// TIA Portal V17 export
// export: Created 2025-06-26T07:49:38.9471019Z, ExportSetting WithDefaults, DisplayName Totally Integrated Automation Portal, DisplayVersion V17 Update 8, DisplayName TIA Portal Openness, DisplayVersion V17 Update 8, DisplayName TIA Portal Version Control Interface, DisplayVersion V17, DisplayName STEP 7 Professional, DisplayVersion V17 Update 8, DisplayName STEP 7 Safety, DisplayVersion V17 Update 6, DisplayName WinCC Advanced, DisplayVersion V17 Update 8
FUNCTION_BLOCK "ControlAlarmHandling"   // FB19, FBD
{ S7_Optimized_Access := 'TRUE' }
VERSION : 0.1
// stored: AutoNumber true, IsIECCheckEnabled false, IsRetainMemResEnabled false, MemoryReserve 0, SetENOAutomatically false, UDAEnableTagReadback false
   VAR
      A1004 { ExternalAccessible := 'False'; ExternalVisible := 'False'; ExternalWritable := 'False'; S7_SetPoint := 'True'} : "fbHMIEvent";
      A2018 { ExternalAccessible := 'False'; ExternalVisible := 'False'; ExternalWritable := 'False'; S7_SetPoint := 'True'} : "fbHighAlarm";
      A2028 { ExternalAccessible := 'False'; ExternalVisible := 'False'; ExternalWritable := 'False'; S7_SetPoint := 'True'} : "fbLowAlarm";
      A2058 { ExternalAccessible := 'False'; ExternalVisible := 'False'; ExternalWritable := 'False'; S7_SetPoint := 'True'} : "fbLowAlarm";
      A2100 { ExternalAccessible := 'False'; ExternalVisible := 'False'; ExternalWritable := 'False'; S7_SetPoint := 'True'} : "fbHighAlarm";
      A2101 { ExternalAccessible := 'False'; ExternalVisible := 'False'; ExternalWritable := 'False'; S7_SetPoint := 'True'} : "fbHighAlarm";
      A2102 { ExternalAccessible := 'False'; ExternalVisible := 'False'; ExternalWritable := 'False'; S7_SetPoint := 'True'} : "fbHighAlarm";
      A2103 { ExternalAccessible := 'False'; ExternalVisible := 'False'; ExternalWritable := 'False'; S7_SetPoint := 'True'} : "fbHighAlarm";
      A2105 { ExternalAccessible := 'False'; ExternalVisible := 'False'; ExternalWritable := 'False'; S7_SetPoint := 'True'} : "fbHighAlarm";
      A2106 { ExternalAccessible := 'False'; ExternalVisible := 'False'; ExternalWritable := 'False'; S7_SetPoint := 'True'} : "fbHighAlarm";
      A2107 { ExternalAccessible := 'False'; ExternalVisible := 'False'; ExternalWritable := 'False'; S7_SetPoint := 'True'} : "fbHighAlarm";
      A2109 { ExternalAccessible := 'False'; ExternalVisible := 'False'; ExternalWritable := 'False'; S7_SetPoint := 'True'} : "fbHighAlarm";
      A2108 { ExternalAccessible := 'False'; ExternalVisible := 'False'; ExternalWritable := 'False'; S7_SetPoint := 'True'} : "fbHighAlarm";
      A2110 { ExternalAccessible := 'False'; ExternalVisible := 'False'; ExternalWritable := 'False'; S7_SetPoint := 'True'} : "fbHighAlarm";
      A2111 { ExternalAccessible := 'False'; ExternalVisible := 'False'; ExternalWritable := 'False'; S7_SetPoint := 'True'} : "fbHighAlarm";
      A2112 { ExternalAccessible := 'False'; ExternalVisible := 'False'; ExternalWritable := 'False'; S7_SetPoint := 'True'} : "fbHighAlarm";
      A2113 { ExternalAccessible := 'False'; ExternalVisible := 'False'; ExternalWritable := 'False'; S7_SetPoint := 'True'} : "fbHighAlarm";
      A2114 { ExternalAccessible := 'False'; ExternalVisible := 'False'; ExternalWritable := 'False'; S7_SetPoint := 'True'} : "fbHighAlarm";
      A2115 { ExternalAccessible := 'False'; ExternalVisible := 'False'; ExternalWritable := 'False'; S7_SetPoint := 'True'} : "fbLowAlarm";
      A2116 { ExternalAccessible := 'False'; ExternalVisible := 'False'; ExternalWritable := 'False'; S7_SetPoint := 'True'} : "fbHighAlarm";
      A2117 { ExternalAccessible := 'False'; ExternalVisible := 'False'; ExternalWritable := 'False'; S7_SetPoint := 'True'} : "fbLowAlarm";
      A2301 { ExternalAccessible := 'False'; ExternalVisible := 'False'; ExternalWritable := 'False'; S7_SetPoint := 'True'} : "fbLowAlarm";
      A2302 { ExternalAccessible := 'False'; ExternalVisible := 'False'; ExternalWritable := 'False'; S7_SetPoint := 'True'} : "fbHighAlarm";
      A2303 { ExternalAccessible := 'False'; ExternalVisible := 'False'; ExternalWritable := 'False'; S7_SetPoint := 'True'} : "fbHighAlarm";
      A2304 { ExternalAccessible := 'False'; ExternalVisible := 'False'; ExternalWritable := 'False'; S7_SetPoint := 'True'} : "fbLowAlarm";
      A2305 { ExternalAccessible := 'False'; ExternalVisible := 'False'; ExternalWritable := 'False'; S7_SetPoint := 'True'} : "fbHighAlarm";
      A2306 { ExternalAccessible := 'False'; ExternalVisible := 'False'; ExternalWritable := 'False'; S7_SetPoint := 'True'} : "fbHighAlarm";
      A2307 { ExternalAccessible := 'False'; ExternalVisible := 'False'; ExternalWritable := 'False'; S7_SetPoint := 'True'} : "fbHMIEvent";
      A2308 { ExternalAccessible := 'False'; ExternalVisible := 'False'; ExternalWritable := 'False'; S7_SetPoint := 'True'} : "fbHighAlarm";
      A3400 { ExternalAccessible := 'False'; ExternalVisible := 'False'; ExternalWritable := 'False'; S7_SetPoint := 'True'} : "fbHMIEvent";
      A9023 { ExternalAccessible := 'False'; ExternalVisible := 'False'; ExternalWritable := 'False'; S7_SetPoint := 'True'} : "fbDeviationAlarm";
      A9024 { S7_SetPoint := 'True'} : "fbDeviationAlarm";
      A9025 { S7_SetPoint := 'True'} : "fbDeviationAlarm";
      A9026 { S7_SetPoint := 'True'} : "fbDeviationAlarm";
      A9027 { S7_SetPoint := 'True'} : "fbDeviationAlarm";
      A9028 { S7_SetPoint := 'True'} : "fbDeviationAlarm";
      A9029 { S7_SetPoint := 'True'} : "fbDeviationAlarm";
      A9030 { S7_SetPoint := 'True'} : "fbDeviationAlarm";
      A9031 { S7_SetPoint := 'True'} : "fbDeviationAlarm";
   END_VAR
   VAR_TEMP   // added for the SCL form of the ladder/FBD networks
      _w1 : Bool;
   END_VAR
BEGIN

REGION Network 1: 1004
   // DISABLED when no connection
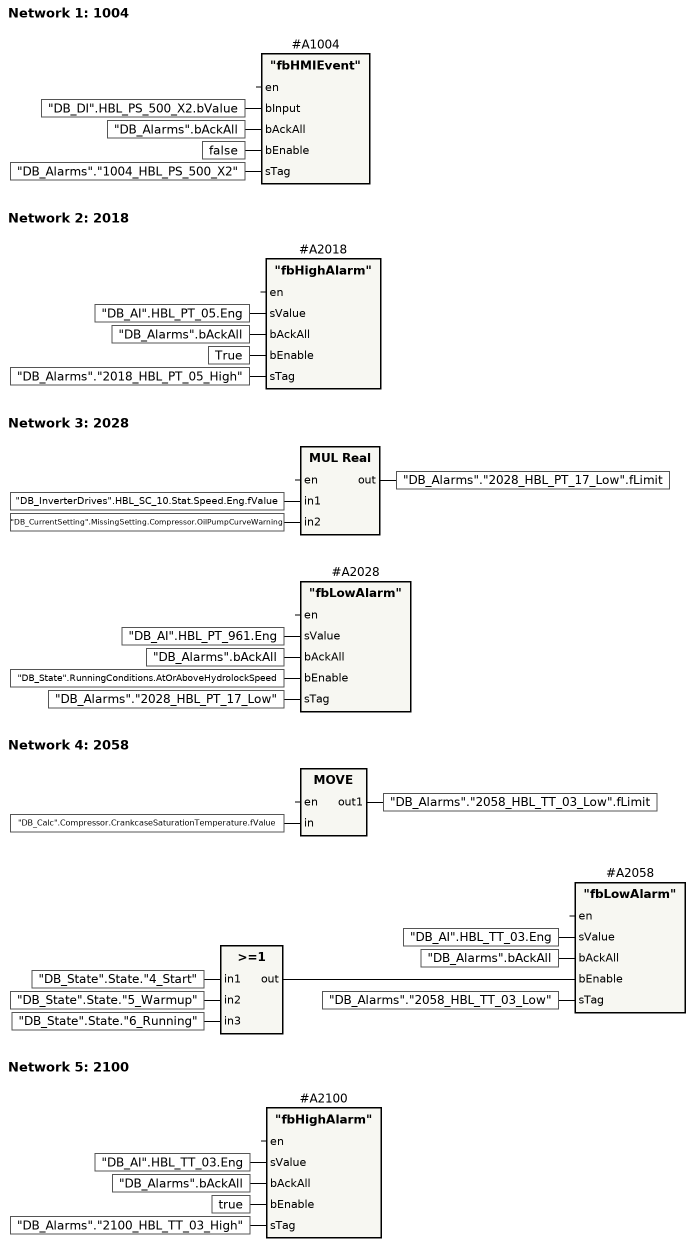
   #A1004(bInput := "DB_DI".HBL_PS_500_X2.bValue,   // "fbHMIEvent"
          bAckAll := "DB_Alarms".bAckAll,
          bEnable := false,
          sTag := "DB_Alarms"."1004_HBL_PS_500_X2");
END_REGION

REGION Network 2: 2018
   #A2018(sValue := "DB_AI".HBL_PT_05.Eng,   // "fbHighAlarm"
          bAckAll := "DB_Alarms".bAckAll,
          bEnable := True,
          sTag := "DB_Alarms"."2018_HBL_PT_05_High");
END_REGION

REGION Network 3: 2028
   // NOTE: alarm limit is dynamic, so don't move it to InitCurrentSettings
   "DB_Alarms"."2028_HBL_PT_17_Low".fLimit := "DB_InverterDrives".HBL_SC_10.Stat.Speed.Eng.fValue * "DB_CurrentSetting".MissingSetting.Compressor.OilPumpCurveWarning;
   #A2028(sValue := "DB_AI".HBL_PT_961.Eng,   // "fbLowAlarm"
          bAckAll := "DB_Alarms".bAckAll,
          bEnable := "DB_State".RunningConditions.AtOrAboveHydrolockSpeed,
          sTag := "DB_Alarms"."2028_HBL_PT_17_Low");
END_REGION

REGION Network 4: 2058
   // NOTE: alarm Low limit is dynamic, so don't move it to InitCurrentSettings
   "DB_Alarms"."2058_HBL_TT_03_Low".fLimit := "DB_Calc".Compressor.CrankcaseSaturationTemperature.fValue;
   #A2058(sValue := "DB_AI".HBL_TT_03.Eng,   // "fbLowAlarm"
          bAckAll := "DB_Alarms".bAckAll,
          bEnable := "DB_State".State."4_Start" OR "DB_State".State."5_Warmup" OR "DB_State".State."6_Running",
          sTag := "DB_Alarms"."2058_HBL_TT_03_Low");
END_REGION

REGION Network 5: 2100
   #A2100(sValue := "DB_AI".HBL_TT_03.Eng,   // "fbHighAlarm"
          bAckAll := "DB_Alarms".bAckAll,
          bEnable := true,
          sTag := "DB_Alarms"."2100_HBL_TT_03_High");
END_REGION

REGION Network 6: 2101
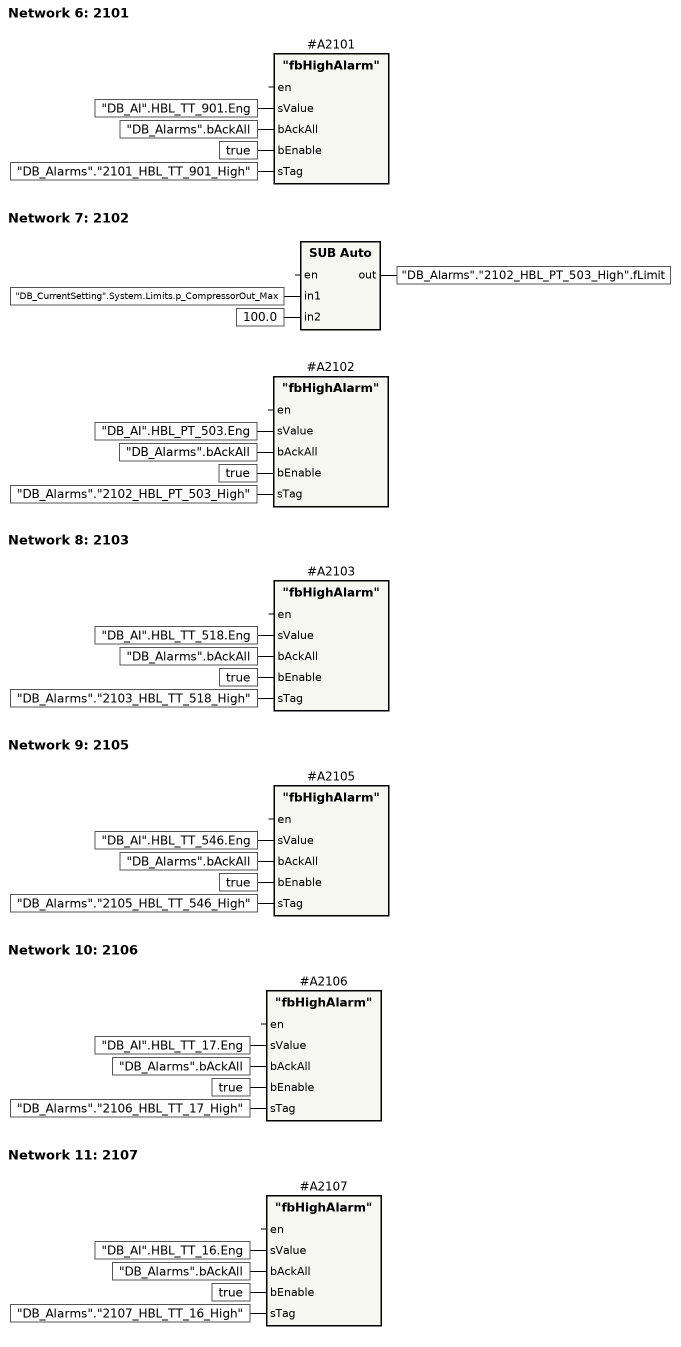
   #A2101(sValue := "DB_AI".HBL_TT_901.Eng,   // "fbHighAlarm"
          bAckAll := "DB_Alarms".bAckAll,
          bEnable := true,
          sTag := "DB_Alarms"."2101_HBL_TT_901_High");
END_REGION

REGION Network 7: 2102
   // Update the alarm limit ALL THE TIME, not just at PLC startup. If the p_CompressorOut_Max value is changed, then this alarms should ALWAYS follow
   "DB_Alarms"."2102_HBL_PT_503_High".fLimit := "DB_CurrentSetting".System.Limits.p_CompressorOut_Max - 100.0;
   #A2102(sValue := "DB_AI".HBL_PT_503.Eng,   // "fbHighAlarm"
          bAckAll := "DB_Alarms".bAckAll,
          bEnable := true,
          sTag := "DB_Alarms"."2102_HBL_PT_503_High");
END_REGION

REGION Network 8: 2103
   #A2103(sValue := "DB_AI".HBL_TT_518.Eng,   // "fbHighAlarm"
          bAckAll := "DB_Alarms".bAckAll,
          bEnable := true,
          sTag := "DB_Alarms"."2103_HBL_TT_518_High");
END_REGION

REGION Network 9: 2105
   #A2105(sValue := "DB_AI".HBL_TT_546.Eng,   // "fbHighAlarm"
          bAckAll := "DB_Alarms".bAckAll,
          bEnable := true,
          sTag := "DB_Alarms"."2105_HBL_TT_546_High");
END_REGION

REGION Network 10: 2106
   #A2106(sValue := "DB_AI".HBL_TT_17.Eng,   // "fbHighAlarm"
          bAckAll := "DB_Alarms".bAckAll,
          bEnable := true,
          sTag := "DB_Alarms"."2106_HBL_TT_17_High");
END_REGION

REGION Network 11: 2107
   #A2107(sValue := "DB_AI".HBL_TT_16.Eng,   // "fbHighAlarm"
          bAckAll := "DB_Alarms".bAckAll,
          bEnable := true,
          sTag := "DB_Alarms"."2107_HBL_TT_16_High");
END_REGION

REGION Network 12: 2108
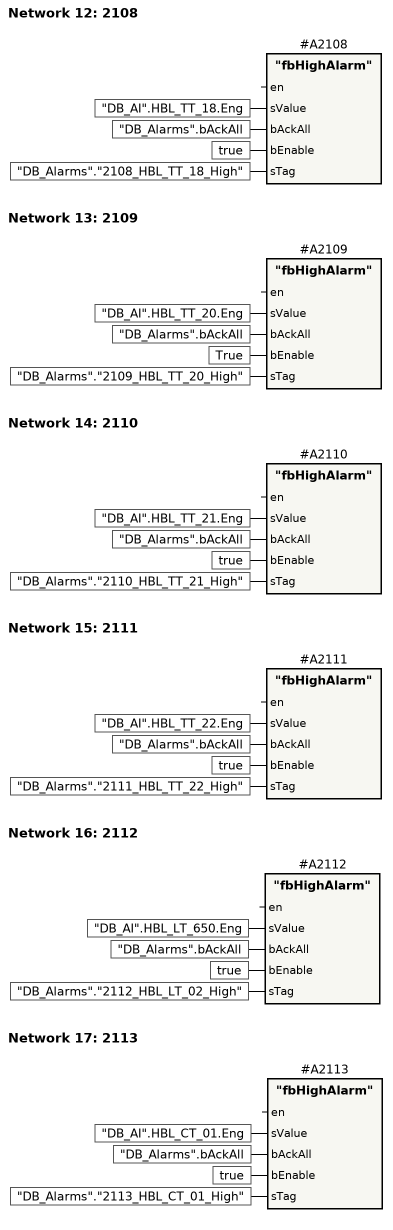
   #A2108(sValue := "DB_AI".HBL_TT_18.Eng,   // "fbHighAlarm"
          bAckAll := "DB_Alarms".bAckAll,
          bEnable := true,
          sTag := "DB_Alarms"."2108_HBL_TT_18_High");
END_REGION

REGION Network 13: 2109
   #A2109(sValue := "DB_AI".HBL_TT_20.Eng,   // "fbHighAlarm"
          bAckAll := "DB_Alarms".bAckAll,
          bEnable := True,
          sTag := "DB_Alarms"."2109_HBL_TT_20_High");
END_REGION

REGION Network 14: 2110
   #A2110(sValue := "DB_AI".HBL_TT_21.Eng,   // "fbHighAlarm"
          bAckAll := "DB_Alarms".bAckAll,
          bEnable := true,
          sTag := "DB_Alarms"."2110_HBL_TT_21_High");
END_REGION

REGION Network 15: 2111
   #A2111(sValue := "DB_AI".HBL_TT_22.Eng,   // "fbHighAlarm"
          bAckAll := "DB_Alarms".bAckAll,
          bEnable := true,
          sTag := "DB_Alarms"."2111_HBL_TT_22_High");
END_REGION

REGION Network 16: 2112
   #A2112(sValue := "DB_AI".HBL_LT_650.Eng,   // "fbHighAlarm"
          bAckAll := "DB_Alarms".bAckAll,
          bEnable := true,
          sTag := "DB_Alarms"."2112_HBL_LT_02_High");
END_REGION

REGION Network 17: 2113
   #A2113(sValue := "DB_AI".HBL_CT_01.Eng,   // "fbHighAlarm"
          bAckAll := "DB_Alarms".bAckAll,
          bEnable := true,
          sTag := "DB_Alarms"."2113_HBL_CT_01_High");
END_REGION

REGION Network 18: 2114
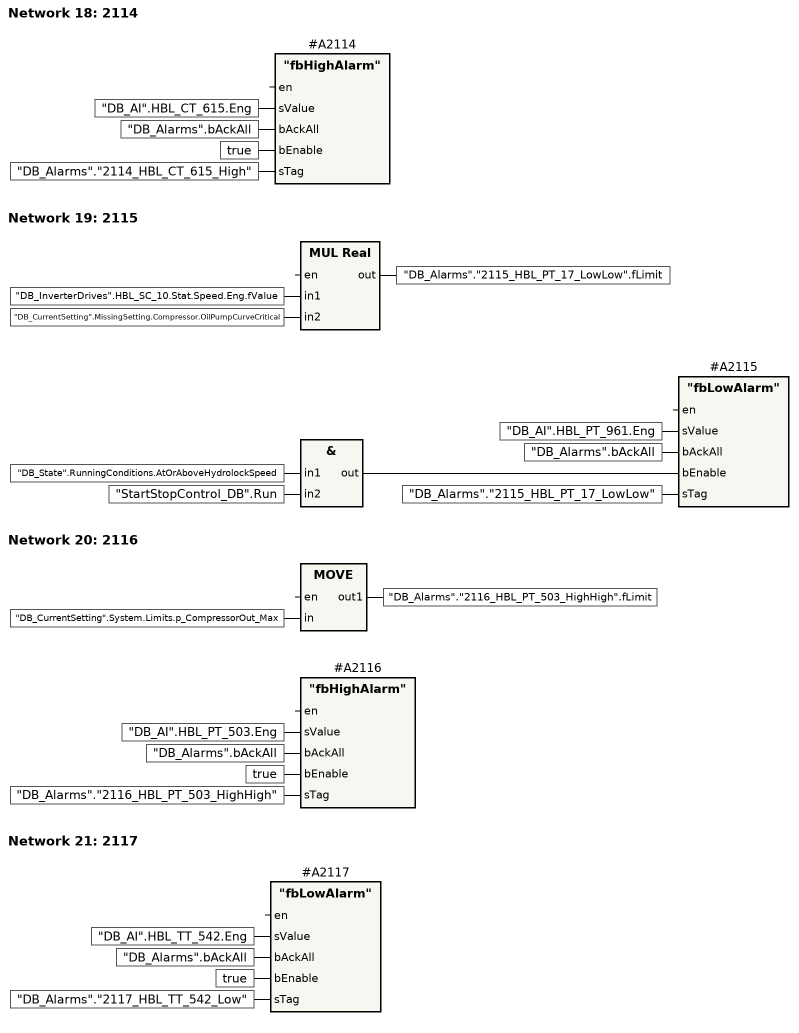
   #A2114(sValue := "DB_AI".HBL_CT_615.Eng,   // "fbHighAlarm"
          bAckAll := "DB_Alarms".bAckAll,
          bEnable := true,
          sTag := "DB_Alarms"."2114_HBL_CT_615_High");
END_REGION

REGION Network 19: 2115
   // NOTE: alarm limit is dynamic, so don't move it to InitCurrentSettings
   "DB_Alarms"."2115_HBL_PT_17_LowLow".fLimit := "DB_InverterDrives".HBL_SC_10.Stat.Speed.Eng.fValue * "DB_CurrentSetting".MissingSetting.Compressor.OilPumpCurveCritical;
   #A2115(sValue := "DB_AI".HBL_PT_961.Eng,   // "fbLowAlarm"
          bAckAll := "DB_Alarms".bAckAll,
          bEnable := "DB_State".RunningConditions.AtOrAboveHydrolockSpeed AND "StartStopControl_DB".Run,
          sTag := "DB_Alarms"."2115_HBL_PT_17_LowLow");
END_REGION

REGION Network 20: 2116
   // Update the alarm limit ALL THE TIME, not just at PLC startup. If the p_CompressorOut_Max value is changed, then this alarms should ALWAYS follow
   "DB_Alarms"."2116_HBL_PT_503_HighHigh".fLimit := "DB_CurrentSetting".System.Limits.p_CompressorOut_Max;
   #A2116(sValue := "DB_AI".HBL_PT_503.Eng,   // "fbHighAlarm"
          bAckAll := "DB_Alarms".bAckAll,
          bEnable := true,
          sTag := "DB_Alarms"."2116_HBL_PT_503_HighHigh");
END_REGION

REGION Network 21: 2117
   #A2117(sValue := "DB_AI".HBL_TT_542.Eng,   // "fbLowAlarm"
          bAckAll := "DB_Alarms".bAckAll,
          bEnable := true,
          sTag := "DB_Alarms"."2117_HBL_TT_542_Low");
END_REGION

REGION Network 22: 2301 & 2302
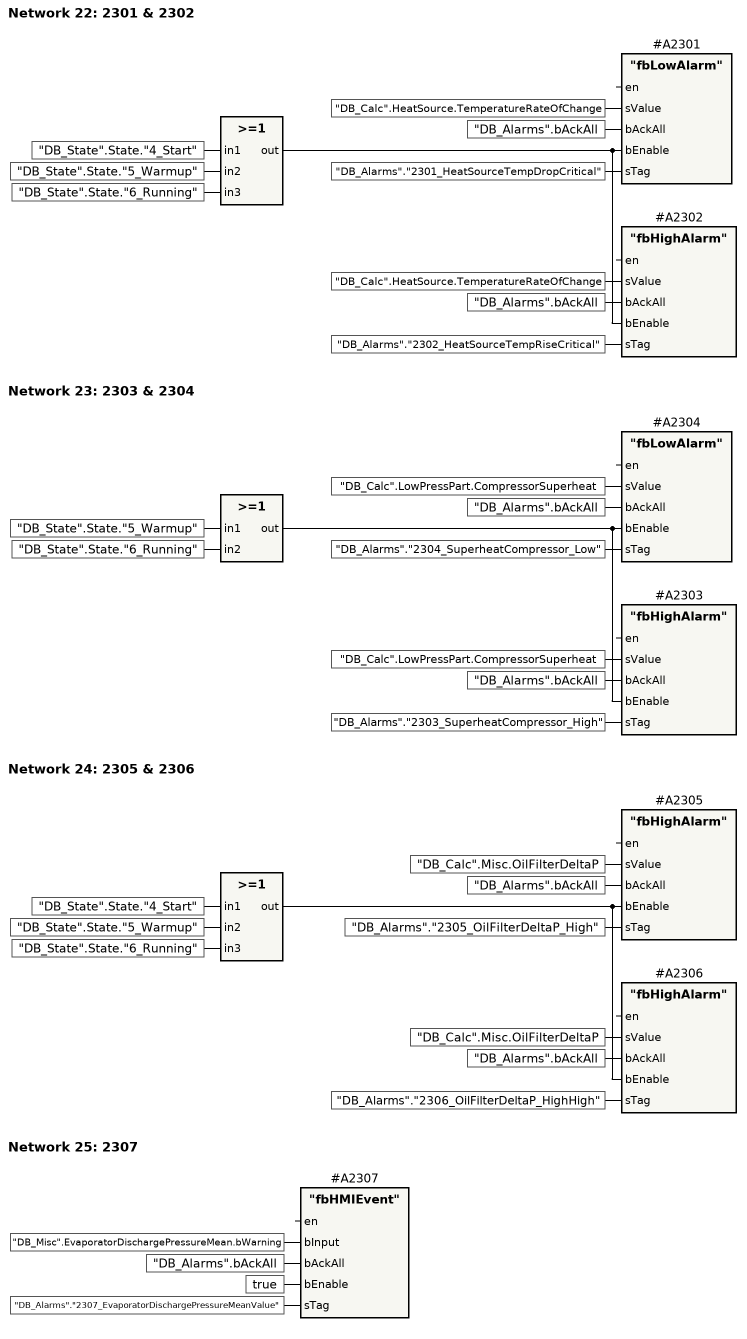
   #_w1 := "DB_State".State."4_Start" OR "DB_State".State."5_Warmup" OR "DB_State".State."6_Running";
   #A2301(sValue := "DB_Calc".HeatSource.TemperatureRateOfChange,   // "fbLowAlarm"
          bAckAll := "DB_Alarms".bAckAll,
          bEnable := #_w1,
          sTag := "DB_Alarms"."2301_HeatSourceTempDropCritical");
   #A2302(sValue := "DB_Calc".HeatSource.TemperatureRateOfChange,   // "fbHighAlarm"
          bAckAll := "DB_Alarms".bAckAll,
          bEnable := #_w1,
          sTag := "DB_Alarms"."2302_HeatSourceTempRiseCritical");
END_REGION

REGION Network 23: 2303 & 2304
   #_w1 := "DB_State".State."5_Warmup" OR "DB_State".State."6_Running";
   #A2304(sValue := "DB_Calc".LowPressPart.CompressorSuperheat,   // "fbLowAlarm"
          bAckAll := "DB_Alarms".bAckAll,
          bEnable := #_w1,
          sTag := "DB_Alarms"."2304_SuperheatCompressor_Low");
   #A2303(sValue := "DB_Calc".LowPressPart.CompressorSuperheat,   // "fbHighAlarm"
          bAckAll := "DB_Alarms".bAckAll,
          bEnable := #_w1,
          sTag := "DB_Alarms"."2303_SuperheatCompressor_High");
END_REGION

REGION Network 24: 2305 & 2306
   #_w1 := "DB_State".State."4_Start" OR "DB_State".State."5_Warmup" OR "DB_State".State."6_Running";
   #A2305(sValue := "DB_Calc".Misc.OilFilterDeltaP,   // "fbHighAlarm"
          bAckAll := "DB_Alarms".bAckAll,
          bEnable := #_w1,
          sTag := "DB_Alarms"."2305_OilFilterDeltaP_High");
   #A2306(sValue := "DB_Calc".Misc.OilFilterDeltaP,   // "fbHighAlarm"
          bAckAll := "DB_Alarms".bAckAll,
          bEnable := #_w1,
          sTag := "DB_Alarms"."2306_OilFilterDeltaP_HighHigh");
END_REGION

REGION Network 25: 2307
   #A2307(bInput := "DB_Misc".EvaporatorDischargePressureMean.bWarning,   // "fbHMIEvent"
          bAckAll := "DB_Alarms".bAckAll,
          bEnable := true,
          sTag := "DB_Alarms"."2307_EvaporatorDischargePressureMeanValue");
END_REGION

REGION Network 26: 2308
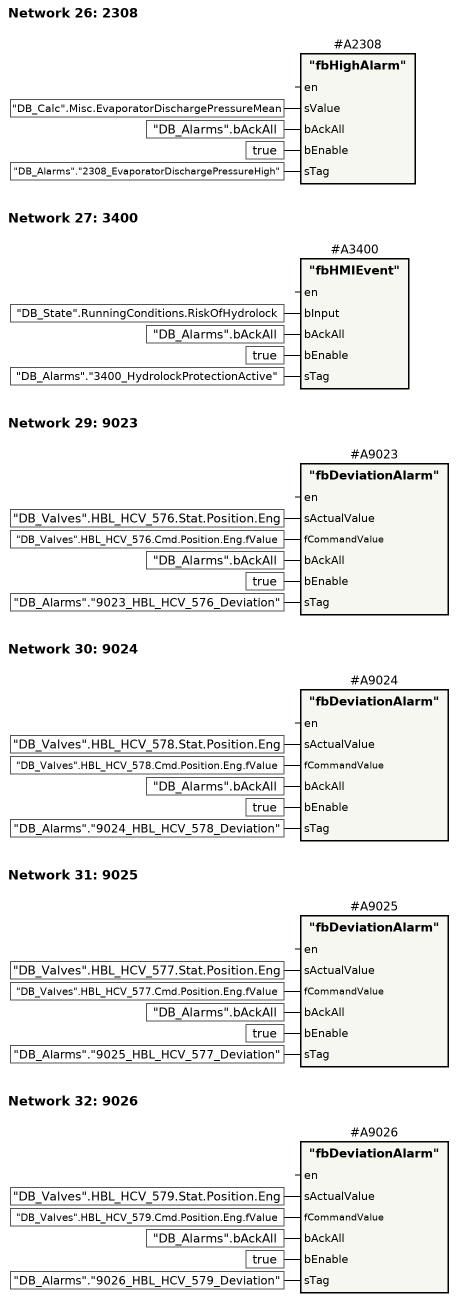
   #A2308(sValue := "DB_Calc".Misc.EvaporatorDischargePressureMean,   // "fbHighAlarm"
          bAckAll := "DB_Alarms".bAckAll,
          bEnable := true,
          sTag := "DB_Alarms"."2308_EvaporatorDischargePressureHigh");
END_REGION

REGION Network 27: 3400
   #A3400(bInput := "DB_State".RunningConditions.RiskOfHydrolock,   // "fbHMIEvent"
          bAckAll := "DB_Alarms".bAckAll,
          bEnable := true,
          sTag := "DB_Alarms"."3400_HydrolockProtectionActive");
END_REGION

REGION Network 28 (SCL): 9023 old
   // This is a deviation alarm, for which a dedicated type does not exist. So we make one here for now with hardocded limits.
   (*
   #A9023(bAckAll := "DB_Alarms".bAckAll, 
           bInput := (ABS(IN := "DB_Valves".HBL_HCV_576.Stat.Position.Eng.fValue -"DB_Valves".HBL_HCV_576.Cmd.Position.Eng.fValue) > 4) OR 
                     ("DB_Valves".HBL_HCV_576.Cmd.Position.Eng.fValue <= 0 AND "DB_Valves".HBL_HCV_576.Stat.Position.Eng.fValue <2),
           sTag := "DB_Alarms"."9023_ExpansionValveDeviation");

   *)
END_REGION

REGION Network 29: 9023
   #A9023(sActualValue := "DB_Valves".HBL_HCV_576.Stat.Position.Eng,   // "fbDeviationAlarm"
          fCommandValue := "DB_Valves".HBL_HCV_576.Cmd.Position.Eng.fValue,
          bAckAll := "DB_Alarms".bAckAll,
          bEnable := true,
          sTag := "DB_Alarms"."9023_HBL_HCV_576_Deviation");
END_REGION

REGION Network 30: 9024
   #A9024(sActualValue := "DB_Valves".HBL_HCV_578.Stat.Position.Eng,   // "fbDeviationAlarm"
          fCommandValue := "DB_Valves".HBL_HCV_578.Cmd.Position.Eng.fValue,
          bAckAll := "DB_Alarms".bAckAll,
          bEnable := true,
          sTag := "DB_Alarms"."9024_HBL_HCV_578_Deviation");
END_REGION

REGION Network 31: 9025
   #A9025(sActualValue := "DB_Valves".HBL_HCV_577.Stat.Position.Eng,   // "fbDeviationAlarm"
          fCommandValue := "DB_Valves".HBL_HCV_577.Cmd.Position.Eng.fValue,
          bAckAll := "DB_Alarms".bAckAll,
          bEnable := true,
          sTag := "DB_Alarms"."9025_HBL_HCV_577_Deviation");
END_REGION

REGION Network 32: 9026
   #A9026(sActualValue := "DB_Valves".HBL_HCV_579.Stat.Position.Eng,   // "fbDeviationAlarm"
          fCommandValue := "DB_Valves".HBL_HCV_579.Cmd.Position.Eng.fValue,
          bAckAll := "DB_Alarms".bAckAll,
          bEnable := true,
          sTag := "DB_Alarms"."9026_HBL_HCV_579_Deviation");
END_REGION

REGION Network 33: 9027
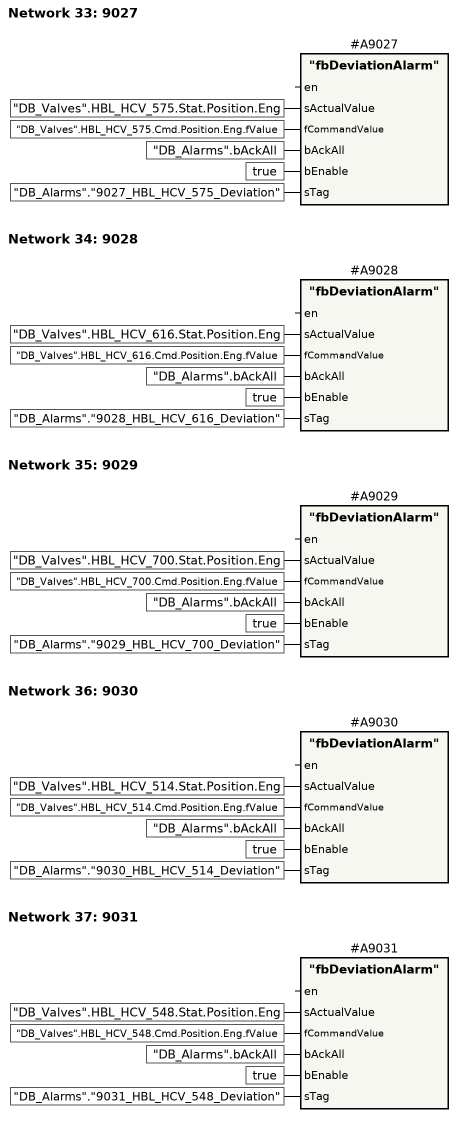
   #A9027(sActualValue := "DB_Valves".HBL_HCV_575.Stat.Position.Eng,   // "fbDeviationAlarm"
          fCommandValue := "DB_Valves".HBL_HCV_575.Cmd.Position.Eng.fValue,
          bAckAll := "DB_Alarms".bAckAll,
          bEnable := true,
          sTag := "DB_Alarms"."9027_HBL_HCV_575_Deviation");
END_REGION

REGION Network 34: 9028
   #A9028(sActualValue := "DB_Valves".HBL_HCV_616.Stat.Position.Eng,   // "fbDeviationAlarm"
          fCommandValue := "DB_Valves".HBL_HCV_616.Cmd.Position.Eng.fValue,
          bAckAll := "DB_Alarms".bAckAll,
          bEnable := true,
          sTag := "DB_Alarms"."9028_HBL_HCV_616_Deviation");
END_REGION

REGION Network 35: 9029
   #A9029(sActualValue := "DB_Valves".HBL_HCV_700.Stat.Position.Eng,   // "fbDeviationAlarm"
          fCommandValue := "DB_Valves".HBL_HCV_700.Cmd.Position.Eng.fValue,
          bAckAll := "DB_Alarms".bAckAll,
          bEnable := true,
          sTag := "DB_Alarms"."9029_HBL_HCV_700_Deviation");
END_REGION

REGION Network 36: 9030
   #A9030(sActualValue := "DB_Valves".HBL_HCV_514.Stat.Position.Eng,   // "fbDeviationAlarm"
          fCommandValue := "DB_Valves".HBL_HCV_514.Cmd.Position.Eng.fValue,
          bAckAll := "DB_Alarms".bAckAll,
          bEnable := true,
          sTag := "DB_Alarms"."9030_HBL_HCV_514_Deviation");
END_REGION

REGION Network 37: 9031
   #A9031(sActualValue := "DB_Valves".HBL_HCV_548.Stat.Position.Eng,   // "fbDeviationAlarm"
          fCommandValue := "DB_Valves".HBL_HCV_548.Cmd.Position.Eng.fValue,
          bAckAll := "DB_Alarms".bAckAll,
          bEnable := true,
          sTag := "DB_Alarms"."9031_HBL_HCV_548_Deviation");
END_REGION
END_FUNCTION_BLOCK
